FUNCTION_BLOCK MTankOut (* Basic Function Block Type *)
  (* Standard: 61499-2 *)
  (* Version 0.0, 2019-06-19, 4DIAC-IDE, 4DIAC-Consortium *)
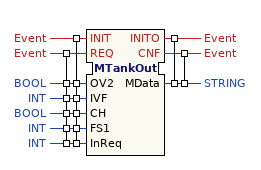
  EVENT_INPUT
    INIT WITH IVF, InReq, FS1, CH, OV2; (* Initialization Request *)
    REQ WITH IVF, InReq, FS1, CH, OV2; (* Normal Execution Request *)
  END_EVENT
  EVENT_OUTPUT
    INITO WITH MData; (* Initialization Confirm *)
    CNF WITH MData; (* Execution Confirmation *)
  END_EVENT
  VAR_INPUT
    OV2 : BOOL;
    IVF : INT;
    CH : BOOL;
    FS1 : INT;
    InReq : INT;
  END_VAR
  VAR_OUTPUT
    MData : STRING; (* Output event qualifier *)
  END_VAR
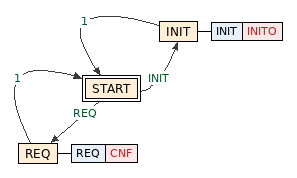
  EC_STATES
    START; (* Initial State *)
    INIT : INIT -> INITO; (* Initialization *)
    REQ : REQ -> CNF; (* Normal execution *)
  END_STATES
  EC_TRANSITIONS
    START TO INIT := INIT;
    INIT TO START := 1;
    START TO REQ := REQ;
    REQ TO START := 1;
  END_TRANSITIONS
  ALGORITHM INIT IN ST: (* Initialization algorithm *)

  END_ALGORITHM
  ALGORITHM REQ IN ST: (* Normally executed algorithm *)
MData := "IEC";
  END_ALGORITHM
END_FUNCTION_BLOCK
